FUNCTION_BLOCK GritScreenLogic_HMI (* Service Interface Function Block Type *)
  (* Standard: 61499-2 *)
  (* Version 0.0, 6/15/2026, Schneider Electric, template *)
  PACKAGE SE.Nereda;
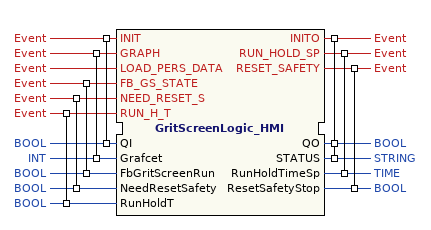
  EVENT_INPUT
    INIT WITH QI;
    GRAPH WITH Grafcet;
    LOAD_PERS_DATA;
    FB_GS_STATE WITH FbGritScreenRun;
    NEED_RESET_S WITH NeedResetSafety;
    RUN_H_T WITH RunHoldT;
  END_EVENT
  EVENT_OUTPUT
    INITO WITH QO, STATUS;
    RUN_HOLD_SP WITH RunHoldTimeSp;
    RESET_SAFETY WITH ResetSafetyStop;
  END_EVENT
  VAR_INPUT
    QI : BOOL;
    Grafcet : INT;
    FbGritScreenRun : BOOL;
    NeedResetSafety : BOOL;
    RunHoldT : BOOL;
  END_VAR
  VAR_OUTPUT
    QO : BOOL; (* Event Output Qualifier *)
    STATUS : STRING; (* Service Status *)
    RunHoldTimeSp : TIME;
    ResetSafetyStop : BOOL;
  END_VAR
  SERVICE /
    SEQUENCE 
    END_SEQUENCE
  END_SERVICE
END_FUNCTION_BLOCK
